// TIA Portal project "2022.06.02_电机顺停" (V17)

(* hardware
DEVICE "S7-1200 station_1"  S7-1200 Station
   slot 0: "Rack_0"  S7-1200 Rack  Rack  V1.0
   slot 1: "PLC_1"  CPU 1212C DC/DC/DC  6ES7 212-1AE40-0XB0  V4.5
*)

// ===== PLC "PLC_1"  CPU 1212C DC/DC/DC =====

VAR_GLOBAL   // PLC tag table "默认变量表"
   "1号启动" AT %I0.0 : Bool;
   "1号电机" AT %Q0.0 : Bool;
   "2号启动" AT %I0.1 : Bool;
   "2号电机" AT %Q0.1 : Bool;
   "2号停止" AT %I0.2 : Bool;
   "1号停止" AT %I0.3 : Bool;
   "中继" AT %M0.0 : Bool;
END_VAR

FUNCTION "电机顺启2" : Void   // FC1, LAD
{ S7_Optimized_Access := 'TRUE' }
VERSION : 0.1
BEGIN

REGION Network 1
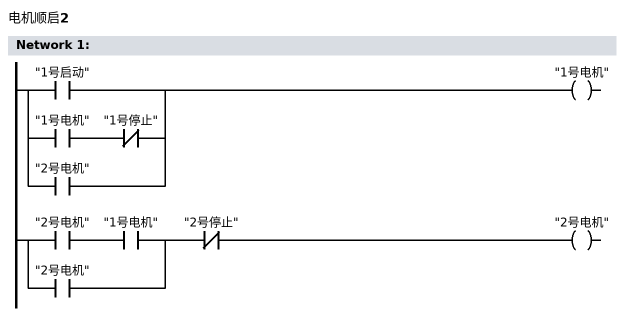
   RUNG wire#powerrail
      Contact( "1号启动" )
      wire#w1
      Coil( "1号电机" )
   END_RUNG
   RUNG wire#powerrail
      Contact( "1号电机" )
      I_Contact( "1号停止" )
   END_RUNG wire#w1
   RUNG wire#powerrail
      Contact( "2号电机" )
   END_RUNG wire#w1
   RUNG wire#powerrail
      Contact( "2号电机" )
      Contact( "1号电机" )
      wire#w2
      I_Contact( "2号停止" )
      Coil( "2号电机" )
   END_RUNG
   RUNG wire#powerrail
      Contact( "2号电机" )
   END_RUNG wire#w2
   // the same network as SCL:
   "1号电机" := "1号启动" OR ("1号电机" AND NOT "1号停止") OR "2号电机";
   "2号电机" := (("2号电机" AND "1号电机") OR "2号电机") AND NOT "2号停止";
END_REGION
END_FUNCTION

ORGANIZATION_BLOCK "Main"   // OB1, LAD, ProgramCycle
TITLE = "Main Program Sweep (Cycle)"
{ S7_Optimized_Access := 'TRUE' }
VERSION : 0.1
   VAR_INPUT
      Initial_Call : Bool;   // Initial call of this OB
      Remanence : Bool;   // =True, if remanent data are available
   END_VAR
BEGIN

REGION Network 1
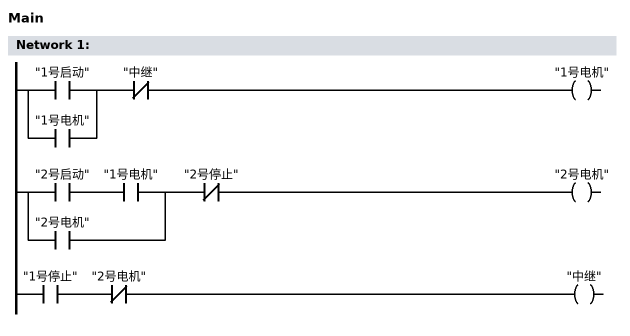
   RUNG wire#powerrail
      Contact( "1号启动" )
      wire#w1
      I_Contact( "中继" )
      Coil( "1号电机" )
   END_RUNG
   RUNG wire#powerrail
      Contact( "1号电机" )
   END_RUNG wire#w1
   RUNG wire#powerrail
      Contact( "2号启动" )
      Contact( "1号电机" )
      wire#w2
      I_Contact( "2号停止" )
      Coil( "2号电机" )
   END_RUNG
   RUNG wire#powerrail
      Contact( "2号电机" )
   END_RUNG wire#w2
   RUNG wire#powerrail
      Contact( "1号停止" )
      I_Contact( "2号电机" )
      Coil( "中继" )
   END_RUNG
   // the same network as SCL:
   "1号电机" := ("1号启动" OR "1号电机") AND NOT "中继";
   "2号电机" := (("2号启动" AND "1号电机") OR "2号电机") AND NOT "2号停止";
   "中继" := "1号停止" AND NOT "2号电机";
END_REGION
END_ORGANIZATION_BLOCK